{attribute addProperty BoxType "EL6201-0000-0017"}
{attribute addProperty Id "Slave_31A_DO0BIT10.125241Slave_31A_DO1BIT10.125242Slave_31A_DO2BIT10.125243Slave_31A_DO3BIT10.125244Slave_31B_DO0BIT10.125245Slave_31B_DO1BIT10.125246Slave_31B_DO2BIT10.125247Slave_31B_DO3BIT10.125248"}
{attribute addProperty CRC "1000640185"}
{attribute addProperty SizeInBites "8"}
{attribute addProperty SizeInBytes "1"}
TYPE Slave_31_Outputs_3BA48EB9 :
STRUCT
	{attribute addProperty Name "Slave_31A_DO0"}
	Slave_31A_DO0 : BIT;
	{attribute addProperty Name "Slave_31A_DO1"}
	Slave_31A_DO1 : BIT;
	{attribute addProperty Name "Slave_31A_DO2"}
	Slave_31A_DO2 : BIT;
	{attribute addProperty Name "Slave_31A_DO3"}
	Slave_31A_DO3 : BIT;
	{attribute addProperty Name "Slave_31B_DO0"}
	Slave_31B_DO0 : BIT;
	{attribute addProperty Name "Slave_31B_DO1"}
	Slave_31B_DO1 : BIT;
	{attribute addProperty Name "Slave_31B_DO2"}
	Slave_31B_DO2 : BIT;
	{attribute addProperty Name "Slave_31B_DO3"}
	Slave_31B_DO3 : BIT;
END_STRUCT
END_TYPE

(* stored: Version 1.2.0.0, ProductVersion 3.1.4024.9
   DUT Slave_31_Outputs_3BA48EB9: Id {cc38cdaf-e195-48ff-b0bf-d6d0b1c5844f} *)
